Fanuc KAREL source: kb00189.KL

PROGRAM KB00189
%STACKSIZE=65535
%PRIORITY=65535
%NOLOCKGROUP
VAR
P1 : STRING[80]
P2 : INTEGER
P3 : INTEGER
RESULT : STRING[80]
BEGIN
P1='A'
P2=1
P3=1
-- UNRESOLVED_PC line 12 opcodes [27 22 2A 22 22 76 75] marker_code=38
END KB00189
